{attribute addProperty BoxType "EL3048-0000-0016"}
{attribute addProperty Id "AI_Standard_ChannelAT %I*ARRAY[0..7] OF AI_Standard_Channel_BC62E3BB576720WcStateAT %I*WcState_98A4DF7520.250InfoDataAT %I*InfoData_BC63D37F80100"}
{attribute addProperty CRC "1840424927"}
{attribute addProperty SizeInBites "658"}
{attribute addProperty SizeInBytes "82.25"}
TYPE EL3048_C9230758 :
STRUCT
	{attribute addProperty Name "AI_Standard_Channel"}
	AI_Standard_Channel : ARRAY[0..7] OF AI_Standard_Channel_BC62E3BB;
	{attribute addProperty Name "WcState"}
	WcState : WcState_98A4DF75;
	{attribute addProperty Name "InfoData"}
	InfoData : InfoData_BC63D37F;
END_STRUCT
END_TYPE

(* stored: Version 1.2.0.0, ProductVersion 3.1.4024.9
   DUT EL3048_C9230758: Id {801983a1-6917-4d5a-8c57-07d1c5cdb16e} *)
